// TIA Portal V16 export
// export: Created 2024-09-05T17:39:22.4057167Z, ExportSetting WithDefaults, DisplayName Totally Integrated Automation Portal, DisplayVersion V16 Update 6, DisplayName TIA Portal Version Control Interface, DisplayVersion V16 Update 2, DisplayName TIA Portal Openness, DisplayVersion V16 Update 6, DisplayName STEP 7 Professional, DisplayVersion V16 Update 6, DisplayName STEP 7 Safety, DisplayVersion V16, DisplayName WinCC Advanced, DisplayVersion V16 Update 6
DATA_BLOCK "setup_DB"   // DB39
VERSION : 0.1
// stored: AutoNumber true, DBAccessibleFromOPCUA true, InstanceOfName setup, InstanceOfType FB
"setup"
   // VAR
   //    alwaysTrue : Bool := TRUE;
   //    counters : Array[0..10] of Int;
   //    maxL : Real;
   //    minL : Real;
   //    maxR : Real;
   //    minR : Real;
   // END_VAR
BEGIN
END_DATA_BLOCK
